FUNCTION F_UpmToDegreePerSec : LREAL
VAR_INPUT
	fValue : LREAL; // 1/min value
END_VAR
VAR
END_VAR

 F_UpmToDegreePerSec := fValue * 6; // 1/min -> °/s => x * 360/60

END_FUNCTION

(* stored: Version 1.1.0.1, ProductVersion 3.1.4024.12
   POU F_UpmToDegreePerSec: Id {8d2b7a62-2cc4-4b6d-a5cf-e7f28b0000cf}, SpecialFunc None *)
